    robot6axis/servo_4/StatusPosDecrease AT 182 : BOOL := false;
    robot6axis/servo_4/displayJauge AT 6454 : REAL := 0.0;
    robot6axis/servo_4/servo_mode/PLC_StatusReady AT 26 : BOOL := true;
    robot6axis/servo_4/servo_mode/PLC_StatusMoved AT 25 : BOOL := false;
    robot6axis/servo_4/servo_mode/PLC_StatusStand AT 24 : BOOL := false;
    robot6axis/servo_4/servo_mode/PLC_ActualPositionAx AT 161 : REAL := 0.0;
    robot6axis/servo_4/servo_mode/PLC_ActualPositionMa AT 48 : REAL := 0.0;
    robot6axis/servo_4/servo_mode/PLC_ActualVelocity AT 47 : REAL := 0.0;
    robot6axis/servo_4/servo_mode/StatusReady AT 266 : BOOL := true;
    robot6axis/servo_4/servo_mode/StatusMoved AT 267 : BOOL := false;
    robot6axis/servo_4/servo_mode/StatusStand AT 268 : BOOL := false;
    robot6axis/servo_4/servo_mode/ActualPositionMa AT 6824 : REAL := 0.0;
    robot6axis/servo_4/servo_mode/ActualVelocity AT 6825 : REAL := 0.0;
    robot6axis/servo_4/servo_mode/MaximumVelocity AT 6826 : REAL := 0.0;
    robot6axis/servo_4/servo_mode/physicalPosInit AT 6461 : REAL := 0.0;
    robot6axis/servo_4/servo_mode/ActualPositionAx AT 6463 : REAL := 0.0;
    robot6axis/servo_4/servo_mode/StatusReady_o AT 186 : BOOL := true;
    robot6axis/servo_4/servo_mode/StatusMoved_o AT 185 : BOOL := false;
    robot6axis/servo_4/servo_mode/StatusStand_o AT 184 : BOOL := false;
    robot6axis/servo_4/servo_mode/ActualPositionAx_o AT 6566 : REAL := 0.0;
    robot6axis/servo_4/servo_mode/ActualPositionMa_o AT 6456 : REAL := 0.0;
    robot6axis/servo_4/servo_mode/ActualVelocity_o AT 39 : REAL := 0.0;
    robot6axis/servo_4/servo_mode/MaximumVelocity_o AT 6455 : REAL := 0.0;
    robot6axis/servo_4/servo_mode/StatusPosIncrease_o AT 183 : BOOL := false;
    robot6axis/servo_4/servo_mode/StatusPosDecrease_o AT 182 : BOOL := false;
    robot6axis/servo_4/servo_mode/displayJauge_o AT 6454 : REAL := 0.0;
    robot6axis/servo_4/servo_mode/PLCMode AT 273 : BOOL := false;
    robot6axis/servo_4/servo_mode/PLCMode1 AT 274 : BOOL := false;
    robot6axis/servo_4/servo_mode/initDone AT 275 : BOOL := false;
    robot6axis/servo_4/servo_mode/displayPosMin AT 6829 : REAL := 0.0;
    robot6axis/servo_4/servo_mode/displayPosMax AT 6830 : REAL := 0.0;
    robot6axis/servo_4/servo_mode/PLC_ActualPositionAx1 AT 6831 : REAL := 0.0;
    robot6axis/servo_4/servo_mode/PLC_ActualVelocity1 AT 6832 : REAL := 0.0;
    robot6axis/servo_4/servo_mode/ActualPositionAx1 AT 6833 : REAL := 0.0;
    robot6axis/servo_4/servo_mode/ActualVelocity1 AT 6834 : REAL := 0.0;
    robot6axis/servo_4/servo_mode/offsetAxToMa AT 6835 : REAL := 0.0;
    robot6axis/servo_4/servo_mode/offsetAxToMa1 AT 6836 : REAL := 0.0;
    robot6axis/servo_4/servo_mode/ActualPositionMa_o1 AT 6837 : REAL := 0.0;
    robot6axis/servo_4/servo_control/HomeCmd AT 56 : BOOL := false;
    robot6axis/servo_4/servo_control/MoveVelCmd AT 55 : BOOL := false;
    robot6axis/servo_4/servo_control/MoveAbsCmd AT 54 : BOOL := false;
    robot6axis/servo_4/servo_control/MoveVel1ManualCmd AT 53 : BOOL := false;
    robot6axis/servo_4/servo_control/MoveVel2ManualCmd AT 52 : BOOL := false;
    robot6axis/servo_4/servo_control/MoveAbs1ManualCmd AT 51 : BOOL := false;
    robot6axis/servo_4/servo_control/MoveAbs2ManualCmd AT 50 : BOOL := false;
    robot6axis/servo_4/servo_control/StopCmd AT 14 : BOOL := false;
    robot6axis/servo_4/servo_control/MovePosition AT 69 : REAL := 0.0;
    robot6axis/servo_4/servo_control/MoveSpeed AT 68 : REAL := 100.0;
    robot6axis/servo_4/servo_control/MoveAcceleration AT 67 : REAL := 100.0;
    robot6axis/servo_4/servo_control/MoveDeceleration AT 66 : REAL := 100.0;
    robot6axis/servo_4/servo_control/offsetAxToMa AT 65 : REAL := 0.0;
    robot6axis/servo_4/servo_control/physicalPosInit AT 6461 : REAL := 0.0;
    robot6axis/servo_4/servo_control/MAX_SPEED AT 6460 : REAL(0.0..3.4e+038) := 30.0;
    robot6axis/servo_4/servo_control/status AT 621 : INT := 0;
    robot6axis/servo_4/servo_control/errorFlag AT 620 : INT := 0;
    robot6axis/servo_4/servo_control/IOActualPositionAx AT 6463 : REAL := 0.0;
    robot6axis/servo_4/servo_control/IOVelDone AT 188 : BOOL := false;
    robot6axis/servo_4/servo_control/IOAbsDone AT 187 : BOOL := false;
    robot6axis/servo_4/servo_control/IOActualVelocity AT 6462 : REAL := 0.0;
    robot6axis/servo_4/servo_control/OperationMode AT 655 : INT := 0;
    robot6axis/servo_4/servo_control/StatusReady AT 266 : BOOL := true;
    robot6axis/servo_4/servo_control/StatusMove AT 267 : BOOL := false;
    robot6axis/servo_4/servo_control/StatusStand AT 268 : BOOL := false;
    robot6axis/servo_4/servo_control/ActualPositionMa AT 6824 : REAL := 0.0;
    robot6axis/servo_4/servo_control/ActualVelocity AT 6825 : REAL := 0.0;
    robot6axis/servo_4/servo_control/MaximumVelocity AT 6826 : REAL := 0.0;
    robot6axis/servo_4/servo_control/VelEnabled AT 269 : BOOL := false;
    robot6axis/servo_4/servo_control/VelCmd AT 270 : BOOL := false;
    robot6axis/servo_4/servo_control/PosEnabled AT 271 : BOOL := false;
    robot6axis/servo_4/servo_control/PosCmd AT 272 : BOOL := false;
    robot6axis/servo_4/servo_control/Position AT 6828 : REAL := 0.0;
    robot6axis/servo_4/servo_control/Speed AT 6827 : REAL := 0.0;
    robot6axis/servo_4/servo_control/ManualMode AT 656 : INT := 0;
    robot6axis/servo_4/servo_control/initDone AT 276 : BOOL := false;
    robot6axis/servo_4/servo_control/ActualPositionMa1 AT 6838 : REAL := 0.0;
    robot6axis/servo_4/servo_control/offsetAxToMa1 AT 6839 : REAL := 0.0;
    robot6axis/servo_4/servo_control/HOME_POSITION AT 6840 : REAL := 100.0;
    robot6axis/servo_4/servo_control/MANUAL_POSITION1 AT 6841 : REAL := 0.0;
    robot6axis/servo_4/servo_control/MANUAL_POSITION2 AT 6842 : REAL := 150.0;
    robot6axis/servo_4/servo_control/MANUAL_SPEED1 AT 6843 : REAL := -100.0;
    robot6axis/servo_4/servo_control/MANUAL_SPEED2 AT 6844 : REAL := 100.0;
    robot6axis/servo_4/servo_control/MANUAL_SPEED AT 6845 : REAL := 100.0;
    robot6axis/servo_4/servo_velocity/MoveVelEnable AT 269 : BOOL := false;
    robot6axis/servo_4/servo_velocity/MoveVelStart AT 270 : BOOL := false;
    robot6axis/servo_4/servo_velocity/MoveSpeed AT 6827 : REAL := 0.0;
    robot6axis/servo_4/servo_velocity/MoveAcceleration AT 67 : REAL := 100.0;
    robot6axis/servo_4/servo_velocity/MoveDeceleration AT 66 : REAL := 100.0;
    robot6axis/servo_4/servo_velocity/MAX_SPEED AT 6460 : REAL(0.0..3.4e+038) := 30.0;
    robot6axis/servo_4/servo_velocity/MAX_ACCEL AT 6459 : REAL(0.0..3.4e+038) := 1500.0;
    robot6axis/servo_4/servo_velocity/MAX_DECEL AT 6458 : REAL(0.0..3.4e+038) := 1500.0;
    robot6axis/servo_4/servo_velocity/MODULO_LENGTH AT 6457 : REAL := 0.0;
    robot6axis/servo_4/servo_velocity/status AT 621 : INT := 0;
    robot6axis/servo_4/servo_velocity/errorFlag AT 620 : INT := 0;
    robot6axis/servo_4/servo_velocity/MoveVelDone AT 188 : BOOL := false;
    robot6axis/servo_4/servo_velocity/ActualPositionAx AT 6463 : REAL := 0.0;
    robot6axis/servo_4/servo_velocity/ActualVelocity AT 6462 : REAL := 0.0;
    robot6axis/servo_4/servo_velocity/firstStep AT 277 : BOOL := true;
    robot6axis/servo_4/servo_velocity/stepDone AT 278 : BOOL := false;
    robot6axis/servo_4/servo_velocity/currentTime AT 6846 : REAL := 0.0;
    robot6axis/servo_4/servo_velocity/MoveSpeed1 AT 6847 : REAL := 0.0;
    robot6axis/servo_4/servo_velocity/acceleration AT 6848 : REAL := 0.0;
    robot6axis/servo_4/servo_velocity/deceleration AT 6849 : REAL := 0.0;
    robot6axis/servo_4/servo_velocity/orderSpeed AT 6850 : REAL := 0.0;
    robot6axis/servo_4/servo_velocity/endChangeSpeed AT 6851 : REAL := 0.0;
    robot6axis/servo_4/servo_velocity/accelDecelChangeSpeed AT 6852 : REAL := 0.0;
    robot6axis/servo_4/servo_velocity/ActualVelocity1 AT 6853 : REAL := 0.0;
    robot6axis/servo_4/servo_velocity/speedChanged AT 279 : BOOL := false;
    robot6axis/servo_4/servo_position/MoveAbsEnable AT 271 : BOOL := false;
    robot6axis/servo_4/servo_position/MoveAbsStart AT 272 : BOOL := false;
    robot6axis/servo_4/servo_position/MovePosition AT 6828 : REAL := 0.0;
    robot6axis/servo_4/servo_position/MoveSpeed AT 6827 : REAL := 0.0;
    robot6axis/servo_4/servo_position/MoveAcceleration AT 67 : REAL := 100.0;
    robot6axis/servo_4/servo_position/MoveDeceleration AT 66 : REAL := 100.0;
    robot6axis/servo_4/servo_position/MAX_SPEED AT 6460 : REAL(0.0..3.4e+038) := 30.0;
    robot6axis/servo_4/servo_position/MAX_ACCEL AT 6459 : REAL(0.0..3.4e+038) := 1500.0;
    robot6axis/servo_4/servo_position/MAX_DECEL AT 6458 : REAL(0.0..3.4e+038) := 1500.0;
    robot6axis/servo_4/servo_position/MODULO_LENGTH AT 6457 : REAL := 0.0;
    robot6axis/servo_4/servo_position/status AT 621 : INT := 0;
    robot6axis/servo_4/servo_position/errorFlag AT 620 : INT := 0;
    robot6axis/servo_4/servo_position/MoveAbsDone AT 187 : BOOL := false;
    robot6axis/servo_4/servo_position/ActualPositionAx AT 6463 : REAL := 0.0;
    robot6axis/servo_4/servo_position/ActualVelocity AT 6462 : REAL := 0.0;
    robot6axis/servo_4/servo_position/firstStep AT 280 : BOOL := true;
    robot6axis/servo_4/servo_position/stepDone AT 281 : BOOL := false;
    robot6axis/servo_4/servo_position/timeToStop AT 6854 : REAL := 0.0;
    robot6axis/servo_4/servo_position/distanceToStop AT 6855 : REAL := 0.0;
    robot6axis/servo_4/servo_position/distance AT 6856 : REAL := 0.0;
    robot6axis/servo_4/servo_position/currentTime AT 6857 : REAL := 0.0;
    robot6axis/servo_4/servo_position/currentSpeed1 AT 6858 : REAL := 0.0;
    robot6axis/servo_4/servo_position/targetPosition AT 6859 : REAL := 0.0;
    robot6axis/servo_4/servo_position/ActualPositionAx1 AT 6860 : REAL := 0.0;
    robot6axis/servo_4/servo_position/acceleration AT 6861 : REAL := 0.0;
    robot6axis/servo_4/servo_position/deceleration AT 6862 : REAL := 0.0;
    robot6axis/servo_4/servo_position/orderSpeed AT 6863 : REAL := 0.0;
    robot6axis/servo_4/servo_position/moveDirection AT 6864 : REAL := 0.0;
    robot6axis/servo_4/servo_position/moveDirection1 AT 6865 : REAL := 0.0;
    robot6axis/servo_4/servo_position/endChangeSpeed AT 6866 : REAL := 0.0;
    robot6axis/servo_4/servo_position/ActualVelocity1 AT 6867 : REAL := 0.0;
    robot6axis/arm4/armOrigin AT 6555 : ARRAY[1..3] OF REAL := [3(0.0)];
    robot6axis/arm4/overallArmQuatInput AT 6560 : ARRAY[1..4] OF REAL := [4(0.0)];
    robot6axis/arm4/structRotVector AT 6449 : ARRAY[1..3] OF REAL := [2(0.0), 1.0];
    robot6axis/arm4/structRotDeg AT 6448 : REAL := 0.0;
    robot6axis/arm4/driveRotVector AT 119 : ARRAY[1..3] OF REAL := [1.0, 2(0.0)];
    robot6axis/arm4/driveRotDeg AT 6566 : REAL := 0.0;
    robot6axis/arm4/ownRotDeg AT 6447 : REAL := 0.0;
    robot6axis/arm4/driveResizeLength AT 6446 : REAL := 0.0;
    robot6axis/arm4/functionActive AT 181 : BOOL := false;
    robot6axis/arm4/armExtrem AT 6567 : ARRAY[1..3] OF REAL := [3(0.0)];
    robot6axis/arm4/overallArmRotOutput AT 6572 : ARRAY[1..4] OF REAL := [4(0.0)];
    robot6axis/arm4/productId AT 619 : DINT := -1;
    robot6axis/arm4/status_act_prod AT 657 : DINT := 0;
    robot6axis/arm4/m11 AT 6868 : REAL := 42.4403;
    robot6axis/arm4/m12 AT 6869 : REAL := 0.0;
    robot6axis/arm4/m13 AT 6870 : REAL := 0.0;
    robot6axis/arm4/m14 AT 6871 : REAL := 11.3174;
    robot6axis/arm4/m21 AT 6872 : REAL := 0.0;
    robot6axis/arm4/m22 AT 6873 : REAL := 31.1229;
    robot6axis/arm4/m23 AT 6874 : REAL := 0.0;
    robot6axis/arm4/m24 AT 6875 : REAL := 100.088;
    robot6axis/arm4/m31 AT 6876 : REAL := 0.0;
    robot6axis/arm4/m32 AT 6877 : REAL := 0.0;
    robot6axis/arm4/m33 AT 6878 : REAL := 9.90274;
    robot6axis/arm4/m34 AT 6879 : REAL := 10.6101;
    robot6axis/arm4/m41 AT 6880 : REAL := 0.0;
    robot6axis/arm4/m42 AT 6881 : REAL := 0.0;
    robot6axis/arm4/m43 AT 6882 : REAL := 0.0;
    robot6axis/arm4/m44 AT 6883 : REAL := 1.0;
    robot6axis/arm4/armLengthCalc AT 6884 : REAL := 0.0;
    robot6axis/arm4/functionActiveLocale AT 282 : BOOL := false;
    robot6axis/arm4/product_id AT 658 : DINT := -1;
    robot6axis/arm4/arm_id AT 659 : DINT := -1;
    robot6axis/arm4/timeToGripParam AT 6885 : REAL := 0.15;
    robot6axis/arm4/armLength AT 6886 : REAL := 202.0;
    robot6axis/arm4/armWidth AT 6887 : REAL := 40.0;
    robot6axis/arm4/armHeight AT 6888 : REAL := 40.0;
    robot6axis/arm4/armType AT 660 : INT := 0;
    robot6axis/servo_5/status AT 618 : INT := 0;
    robot6axis/servo_5/errorFlag AT 617 : INT := 0;
    robot6axis/servo_5/ActualPositionAx1 AT 6445 : REAL := 0.0;
    robot6axis/servo_5/MoveVelDone1 AT 180 : BOOL := false;
    robot6axis/servo_5/ActualVelocity1 AT 6444 : REAL := 0.0;
    robot6axis/servo_5/MoveAbsDone1 AT 179 : BOOL := false;
    robot6axis/servo_5/HomeCmd AT 49 : BOOL := false;
    robot6axis/servo_5/MoveVelCmd AT 48 : BOOL := false;
    robot6axis/servo_5/MoveAbsCmd AT 47 : BOOL := false;
    robot6axis/servo_5/MoveVel1ManualCmd AT 46 : BOOL := false;
    robot6axis/servo_5/MoveVel2ManualCmd AT 45 : BOOL := false;
    robot6axis/servo_5/MoveAbs1ManualCmd AT 44 : BOOL := false;
    robot6axis/servo_5/MoveAbs2ManualCmd AT 43 : BOOL := false;
    robot6axis/servo_5/StopCmd AT 14 : BOOL := false;
    robot6axis/servo_5/MovePosition AT 64 : REAL := 0.0;
    robot6axis/servo_5/MoveSpeed AT 63 : REAL := 100.0;
    robot6axis/servo_5/MoveAcceleration AT 62 : REAL := 100.0;
    robot6axis/servo_5/MoveDeceleration AT 61 : REAL := 100.0;
    robot6axis/servo_5/offsetAxToMa AT 60 : REAL := 0.0;
    robot6axis/servo_5/PLC_StatusReady AT 23 : BOOL := true;
    robot6axis/servo_5/PLC_StatusMoved AT 22 : BOOL := false;
    robot6axis/servo_5/PLC_StatusStand AT 21 : BOOL := false;
    robot6axis/servo_5/PLC_ActualPositionAx AT 162 : REAL := 0.0;
    robot6axis/servo_5/PLC_ActualPositionMa AT 46 : REAL := 0.0;
    robot6axis/servo_5/PLC_ActualVelocity AT 45 : REAL := 0.0;
    robot6axis/servo_5/physicalPosInit AT 6443 : REAL := 0.0;
    robot6axis/servo_5/MAX_SPEED AT 6442 : REAL(0.0..3.4e+038) := 30.0;
    robot6axis/servo_5/MAX_ACCEL AT 6441 : REAL(0.0..3.4e+038) := 1500.0;
    robot6axis/servo_5/MAX_DECEL AT 6440 : REAL(0.0..3.4e+038) := 1500.0;
    robot6axis/servo_5/MODULO_LENGTH AT 6439 : REAL := 0.0;
    robot6axis/servo_5/StatusReady AT 178 : BOOL := true;
    robot6axis/servo_5/StatusMoved AT 177 : BOOL := false;
    robot6axis/servo_5/StatusStand AT 176 : BOOL := false;
    robot6axis/servo_5/ActualPositionAx AT 6578 : REAL := 0.0;
    robot6axis/servo_5/ActualPositionMa AT 6438 : REAL := 0.0;
    robot6axis/servo_5/ActualVelocity AT 38 : REAL := 0.0;
    robot6axis/servo_5/MaximumVelocity AT 6437 : REAL := 0.0;
    robot6axis/servo_5/StatusPosIncrease AT 175 : BOOL := false;
    robot6axis/servo_5/StatusPosDecrease AT 174 : BOOL := false;
    robot6axis/servo_5/displayJauge AT 6436 : REAL := 0.0;
    robot6axis/servo_5/servo_mode/PLC_StatusReady AT 23 : BOOL := true;
    robot6axis/servo_5/servo_mode/PLC_StatusMoved AT 22 : BOOL := false;
    robot6axis/servo_5/servo_mode/PLC_StatusStand AT 21 : BOOL := false;
    robot6axis/servo_5/servo_mode/PLC_ActualPositionAx AT 162 : REAL := 0.0;
    robot6axis/servo_5/servo_mode/PLC_ActualPositionMa AT 46 : REAL := 0.0;
    robot6axis/servo_5/servo_mode/PLC_ActualVelocity AT 45 : REAL := 0.0;
    robot6axis/servo_5/servo_mode/StatusReady AT 283 : BOOL := true;
    robot6axis/servo_5/servo_mode/StatusMoved AT 284 : BOOL := false;
    robot6axis/servo_5/servo_mode/StatusStand AT 285 : BOOL := false;
    robot6axis/servo_5/servo_mode/ActualPositionMa AT 6889 : REAL := 0.0;
    robot6axis/servo_5/servo_mode/ActualVelocity AT 6890 : REAL := 0.0;
    robot6axis/servo_5/servo_mode/MaximumVelocity AT 6891 : REAL := 0.0;
    robot6axis/servo_5/servo_mode/physicalPosInit AT 6443 : REAL := 0.0;
    robot6axis/servo_5/servo_mode/ActualPositionAx AT 6445 : REAL := 0.0;
    robot6axis/servo_5/servo_mode/StatusReady_o AT 178 : BOOL := true;
    robot6axis/servo_5/servo_mode/StatusMoved_o AT 177 : BOOL := false;
    robot6axis/servo_5/servo_mode/StatusStand_o AT 176 : BOOL := false;
    robot6axis/servo_5/servo_mode/ActualPositionAx_o AT 6578 : REAL := 0.0;
    robot6axis/servo_5/servo_mode/ActualPositionMa_o AT 6438 : REAL := 0.0;
    robot6axis/servo_5/servo_mode/ActualVelocity_o AT 38 : REAL := 0.0;
    robot6axis/servo_5/servo_mode/MaximumVelocity_o AT 6437 : REAL := 0.0;
    robot6axis/servo_5/servo_mode/StatusPosIncrease_o AT 175 : BOOL := false;
    robot6axis/servo_5/servo_mode/StatusPosDecrease_o AT 174 : BOOL := false;
    robot6axis/servo_5/servo_mode/displayJauge_o AT 6436 : REAL := 0.0;
    robot6axis/servo_5/servo_mode/PLCMode AT 290 : BOOL := false;
    robot6axis/servo_5/servo_mode/PLCMode1 AT 291 : BOOL := false;
    robot6axis/servo_5/servo_mode/initDone AT 292 : BOOL := false;
    robot6axis/servo_5/servo_mode/displayPosMin AT 6894 : REAL := 0.0;
    robot6axis/servo_5/servo_mode/displayPosMax AT 6895 : REAL := 0.0;
    robot6axis/servo_5/servo_mode/PLC_ActualPositionAx1 AT 6896 : REAL := 0.0;
    robot6axis/servo_5/servo_mode/PLC_ActualVelocity1 AT 6897 : REAL := 0.0;
    robot6axis/servo_5/servo_mode/ActualPositionAx1 AT 6898 : REAL := 0.0;
    robot6axis/servo_5/servo_mode/ActualVelocity1 AT 6899 : REAL := 0.0;
    robot6axis/servo_5/servo_mode/offsetAxToMa AT 6900 : REAL := 0.0;
    robot6axis/servo_5/servo_mode/offsetAxToMa1 AT 6901 : REAL := 0.0;
    robot6axis/servo_5/servo_mode/ActualPositionMa_o1 AT 6902 : REAL := 0.0;
    robot6axis/servo_5/servo_control/HomeCmd AT 49 : BOOL := false;
    robot6axis/servo_5/servo_control/MoveVelCmd AT 48 : BOOL := false;
    robot6axis/servo_5/servo_control/MoveAbsCmd AT 47 : BOOL := false;
    robot6axis/servo_5/servo_control/MoveVel1ManualCmd AT 46 : BOOL := false;
    robot6axis/servo_5/servo_control/MoveVel2ManualCmd AT 45 : BOOL := false;
    robot6axis/servo_5/servo_control/MoveAbs1ManualCmd AT 44 : BOOL := false;
    robot6axis/servo_5/servo_control/MoveAbs2ManualCmd AT 43 : BOOL := false;
    robot6axis/servo_5/servo_control/StopCmd AT 14 : BOOL := false;
    robot6axis/servo_5/servo_control/MovePosition AT 64 : REAL := 0.0;
    robot6axis/servo_5/servo_control/MoveSpeed AT 63 : REAL := 100.0;
    robot6axis/servo_5/servo_control/MoveAcceleration AT 62 : REAL := 100.0;
    robot6axis/servo_5/servo_control/MoveDeceleration AT 61 : REAL := 100.0;
    robot6axis/servo_5/servo_control/offsetAxToMa AT 60 : REAL := 0.0;
    robot6axis/servo_5/servo_control/physicalPosInit AT 6443 : REAL := 0.0;
    robot6axis/servo_5/servo_control/MAX_SPEED AT 6442 : REAL(0.0..3.4e+038) := 30.0;
    robot6axis/servo_5/servo_control/status AT 618 : INT := 0;
    robot6axis/servo_5/servo_control/errorFlag AT 617 : INT := 0;
    robot6axis/servo_5/servo_control/IOActualPositionAx AT 6445 : REAL := 0.0;
    robot6axis/servo_5/servo_control/IOVelDone AT 180 : BOOL := false;
    robot6axis/servo_5/servo_control/IOAbsDone AT 179 : BOOL := false;
    robot6axis/servo_5/servo_control/IOActualVelocity AT 6444 : REAL := 0.0;
    robot6axis/servo_5/servo_control/OperationMode AT 661 : INT := 0;
    robot6axis/servo_5/servo_control/StatusReady AT 283 : BOOL := true;
    robot6axis/servo_5/servo_control/StatusMove AT 284 : BOOL := false;
    robot6axis/servo_5/servo_control/StatusStand AT 285 : BOOL := false;
    robot6axis/servo_5/servo_control/ActualPositionMa AT 6889 : REAL := 0.0;
    robot6axis/servo_5/servo_control/ActualVelocity AT 6890 : REAL := 0.0;
    robot6axis/servo_5/servo_control/MaximumVelocity AT 6891 : REAL := 0.0;
    robot6axis/servo_5/servo_control/VelEnabled AT 286 : BOOL := false;
    robot6axis/servo_5/servo_control/VelCmd AT 287 : BOOL := false;
    robot6axis/servo_5/servo_control/PosEnabled AT 288 : BOOL := false;
    robot6axis/servo_5/servo_control/PosCmd AT 289 : BOOL := false;
    robot6axis/servo_5/servo_control/Position AT 6893 : REAL := 0.0;
    robot6axis/servo_5/servo_control/Speed AT 6892 : REAL := 0.0;
    robot6axis/servo_5/servo_control/ManualMode AT 662 : INT := 0;
    robot6axis/servo_5/servo_control/initDone AT 293 : BOOL := false;
    robot6axis/servo_5/servo_control/ActualPositionMa1 AT 6903 : REAL := 0.0;
    robot6axis/servo_5/servo_control/offsetAxToMa1 AT 6904 : REAL := 0.0;
    robot6axis/servo_5/servo_control/HOME_POSITION AT 6905 : REAL := 100.0;
    robot6axis/servo_5/servo_control/MANUAL_POSITION1 AT 6906 : REAL := 0.0;
    robot6axis/servo_5/servo_control/MANUAL_POSITION2 AT 6907 : REAL := 150.0;
    robot6axis/servo_5/servo_control/MANUAL_SPEED1 AT 6908 : REAL := -100.0;
    robot6axis/servo_5/servo_control/MANUAL_SPEED2 AT 6909 : REAL := 100.0;
    robot6axis/servo_5/servo_control/MANUAL_SPEED AT 6910 : REAL := 100.0;
    robot6axis/servo_5/servo_velocity/MoveVelEnable AT 286 : BOOL := false;
    robot6axis/servo_5/servo_velocity/MoveVelStart AT 287 : BOOL := false;
    robot6axis/servo_5/servo_velocity/MoveSpeed AT 6892 : REAL := 0.0;
    robot6axis/servo_5/servo_velocity/MoveAcceleration AT 62 : REAL := 100.0;
    robot6axis/servo_5/servo_velocity/MoveDeceleration AT 61 : REAL := 100.0;
    robot6axis/servo_5/servo_velocity/MAX_SPEED AT 6442 : REAL(0.0..3.4e+038) := 30.0;
    robot6axis/servo_5/servo_velocity/MAX_ACCEL AT 6441 : REAL(0.0..3.4e+038) := 1500.0;
    robot6axis/servo_5/servo_velocity/MAX_DECEL AT 6440 : REAL(0.0..3.4e+038) := 1500.0;
    robot6axis/servo_5/servo_velocity/MODULO_LENGTH AT 6439 : REAL := 0.0;
    robot6axis/servo_5/servo_velocity/status AT 618 : INT := 0;
    robot6axis/servo_5/servo_velocity/errorFlag AT 617 : INT := 0;
    robot6axis/servo_5/servo_velocity/MoveVelDone AT 180 : BOOL := false;
    robot6axis/servo_5/servo_velocity/ActualPositionAx AT 6445 : REAL := 0.0;
    robot6axis/servo_5/servo_velocity/ActualVelocity AT 6444 : REAL := 0.0;
    robot6axis/servo_5/servo_velocity/firstStep AT 294 : BOOL := true;
    robot6axis/servo_5/servo_velocity/stepDone AT 295 : BOOL := false;
    robot6axis/servo_5/servo_velocity/currentTime AT 6911 : REAL := 0.0;
    robot6axis/servo_5/servo_velocity/MoveSpeed1 AT 6912 : REAL := 0.0;
    robot6axis/servo_5/servo_velocity/acceleration AT 6913 : REAL := 0.0;
    robot6axis/servo_5/servo_velocity/deceleration AT 6914 : REAL := 0.0;
    robot6axis/servo_5/servo_velocity/orderSpeed AT 6915 : REAL := 0.0;
    robot6axis/servo_5/servo_velocity/endChangeSpeed AT 6916 : REAL := 0.0;
    robot6axis/servo_5/servo_velocity/accelDecelChangeSpeed AT 6917 : REAL := 0.0;
    robot6axis/servo_5/servo_velocity/ActualVelocity1 AT 6918 : REAL := 0.0;
    robot6axis/servo_5/servo_velocity/speedChanged AT 296 : BOOL := false;
    robot6axis/servo_5/servo_position/MoveAbsEnable AT 288 : BOOL := false;
    robot6axis/servo_5/servo_position/MoveAbsStart AT 289 : BOOL := false;
    robot6axis/servo_5/servo_position/MovePosition AT 6893 : REAL := 0.0;
    robot6axis/servo_5/servo_position/MoveSpeed AT 6892 : REAL := 0.0;
    robot6axis/servo_5/servo_position/MoveAcceleration AT 62 : REAL := 100.0;
    robot6axis/servo_5/servo_position/MoveDeceleration AT 61 : REAL := 100.0;
    robot6axis/servo_5/servo_position/MAX_SPEED AT 6442 : REAL(0.0..3.4e+038) := 30.0;
    robot6axis/servo_5/servo_position/MAX_ACCEL AT 6441 : REAL(0.0..3.4e+038) := 1500.0;
    robot6axis/servo_5/servo_position/MAX_DECEL AT 6440 : REAL(0.0..3.4e+038) := 1500.0;
    robot6axis/servo_5/servo_position/MODULO_LENGTH AT 6439 : REAL := 0.0;
    robot6axis/servo_5/servo_position/status AT 618 : INT := 0;
    robot6axis/servo_5/servo_position/errorFlag AT 617 : INT := 0;
    robot6axis/servo_5/servo_position/MoveAbsDone AT 179 : BOOL := false;
    robot6axis/servo_5/servo_position/ActualPositionAx AT 6445 : REAL := 0.0;
    robot6axis/servo_5/servo_position/ActualVelocity AT 6444 : REAL := 0.0;
    robot6axis/servo_5/servo_position/firstStep AT 297 : BOOL := true;
    robot6axis/servo_5/servo_position/stepDone AT 298 : BOOL := false;
    robot6axis/servo_5/servo_position/timeToStop AT 6919 : REAL := 0.0;
    robot6axis/servo_5/servo_position/distanceToStop AT 6920 : REAL := 0.0;
    robot6axis/servo_5/servo_position/distance AT 6921 : REAL := 0.0;
    robot6axis/servo_5/servo_position/currentTime AT 6922 : REAL := 0.0;
    robot6axis/servo_5/servo_position/currentSpeed1 AT 6923 : REAL := 0.0;
    robot6axis/servo_5/servo_position/targetPosition AT 6924 : REAL := 0.0;
    robot6axis/servo_5/servo_position/ActualPositionAx1 AT 6925 : REAL := 0.0;
    robot6axis/servo_5/servo_position/acceleration AT 6926 : REAL := 0.0;
    robot6axis/servo_5/servo_position/deceleration AT 6927 : REAL := 0.0;
    robot6axis/servo_5/servo_position/orderSpeed AT 6928 : REAL := 0.0;
    robot6axis/servo_5/servo_position/moveDirection AT 6929 : REAL := 0.0;
    robot6axis/servo_5/servo_position/moveDirection1 AT 6930 : REAL := 0.0;
    robot6axis/servo_5/servo_position/endChangeSpeed AT 6931 : REAL := 0.0;
    robot6axis/servo_5/servo_position/ActualVelocity1 AT 6932 : REAL := 0.0;
    robot6axis/arm5/armOrigin AT 6567 : ARRAY[1..3] OF REAL := [3(0.0)];
    robot6axis/arm5/overallArmQuatInput AT 6572 : ARRAY[1..4] OF REAL := [4(0.0)];
    robot6axis/arm5/structRotVector AT 6431 : ARRAY[1..3] OF REAL := [2(0.0), 1.0];
    robot6axis/arm5/structRotDeg AT 6430 : REAL := 0.0;
    robot6axis/arm5/driveRotVector AT 114 : ARRAY[1..3] OF REAL := [0.0, 1.0, 0.0];
    robot6axis/arm5/driveRotDeg AT 6578 : REAL := 0.0;
    robot6axis/arm5/ownRotDeg AT 6429 : REAL := 0.0;
    robot6axis/arm5/driveResizeLength AT 6428 : REAL := 0.0;
    robot6axis/arm5/functionActive AT 173 : BOOL := false;
    robot6axis/arm5/armExtrem AT 6579 : ARRAY[1..3] OF REAL := [3(0.0)];
    robot6axis/arm5/overallArmRotOutput AT 6584 : ARRAY[1..4] OF REAL := [4(0.0)];
    robot6axis/arm5/productId AT 616 : DINT := -1;
    robot6axis/arm5/status_act_prod AT 663 : DINT := 0;
    robot6axis/arm5/m11 AT 6933 : REAL := 38.1963;
    robot6axis/arm5/m12 AT 6934 : REAL := 0.0;
    robot6axis/arm5/m13 AT 6935 : REAL := 0.0;
    robot6axis/arm5/m14 AT 6936 : REAL := 8.48806;
    robot6axis/arm5/m21 AT 6937 : REAL := 0.0;
    robot6axis/arm5/m22 AT 6938 : REAL := 1.0;
    robot6axis/arm5/m23 AT 6939 : REAL := 0.0;
    robot6axis/arm5/m24 AT 6940 : REAL := 1.0;
    robot6axis/arm5/m31 AT 6941 : REAL := 0.0;
    robot6axis/arm5/m32 AT 6942 : REAL := 0.0;
    robot6axis/arm5/m33 AT 6943 : REAL := 14.1468;
    robot6axis/arm5/m34 AT 6944 : REAL := -10.6101;
    robot6axis/arm5/m41 AT 6945 : REAL := 0.0;
    robot6axis/arm5/m42 AT 6946 : REAL := 0.0;
    robot6axis/arm5/m43 AT 6947 : REAL := 0.0;
    robot6axis/arm5/m44 AT 6948 : REAL := 1.0;
    robot6axis/arm5/armLengthCalc AT 6949 : REAL := 0.0;
    robot6axis/arm5/functionActiveLocale AT 299 : BOOL := false;
    robot6axis/arm5/product_id AT 664 : DINT := -1;
    robot6axis/arm5/arm_id AT 665 : DINT := -1;
    robot6axis/arm5/timeToGripParam AT 6950 : REAL := 0.15;
    robot6axis/arm5/armLength AT 6951 : REAL := 61.0;
    robot6axis/arm5/armWidth AT 6952 : REAL := 40.0;
    robot6axis/arm5/armHeight AT 6953 : REAL := 40.0;
    robot6axis/arm5/armType AT 666 : INT := 0;
    robot6axis/servo_6/status AT 615 : INT := 0;
    robot6axis/servo_6/errorFlag AT 614 : INT := 0;
    robot6axis/servo_6/ActualPositionAx1 AT 6427 : REAL := 0.0;
    robot6axis/servo_6/MoveVelDone1 AT 172 : BOOL := false;
    robot6axis/servo_6/ActualVelocity1 AT 6426 : REAL := 0.0;
    robot6axis/servo_6/MoveAbsDone1 AT 171 : BOOL := false;
    robot6axis/servo_6/HomeCmd AT 42 : BOOL := false;
    robot6axis/servo_6/MoveVelCmd AT 41 : BOOL := false;
    robot6axis/servo_6/MoveAbsCmd AT 40 : BOOL := false;
    robot6axis/servo_6/MoveVel1ManualCmd AT 39 : BOOL := false;
    robot6axis/servo_6/MoveVel2ManualCmd AT 38 : BOOL := false;
    robot6axis/servo_6/MoveAbs1ManualCmd AT 37 : BOOL := false;
    robot6axis/servo_6/MoveAbs2ManualCmd AT 36 : BOOL := false;
    robot6axis/servo_6/StopCmd AT 14 : BOOL := false;
    robot6axis/servo_6/MovePosition AT 59 : REAL := 0.0;
    robot6axis/servo_6/MoveSpeed AT 58 : REAL := 100.0;
    robot6axis/servo_6/MoveAcceleration AT 57 : REAL := 100.0;
    robot6axis/servo_6/MoveDeceleration AT 56 : REAL := 100.0;
    robot6axis/servo_6/offsetAxToMa AT 55 : REAL := 0.0;
    robot6axis/servo_6/PLC_StatusReady AT 20 : BOOL := true;
    robot6axis/servo_6/PLC_StatusMoved AT 19 : BOOL := false;
    robot6axis/servo_6/PLC_StatusStand AT 18 : BOOL := false;
    robot6axis/servo_6/PLC_ActualPositionAx AT 163 : REAL := 0.0;
    robot6axis/servo_6/PLC_ActualPositionMa AT 44 : REAL := 0.0;
    robot6axis/servo_6/PLC_ActualVelocity AT 43 : REAL := 0.0;
    robot6axis/servo_6/physicalPosInit AT 6425 : REAL := 0.0;
    robot6axis/servo_6/MAX_SPEED AT 6424 : REAL(0.0..3.4e+038) := 30.0;
    robot6axis/servo_6/MAX_ACCEL AT 6423 : REAL(0.0..3.4e+038) := 1500.0;
    robot6axis/servo_6/MAX_DECEL AT 6422 : REAL(0.0..3.4e+038) := 1500.0;
    robot6axis/servo_6/MODULO_LENGTH AT 6421 : REAL := 0.0;
    robot6axis/servo_6/StatusReady AT 170 : BOOL := true;
    robot6axis/servo_6/StatusMoved AT 169 : BOOL := false;
    robot6axis/servo_6/StatusStand AT 168 : BOOL := false;
    robot6axis/servo_6/ActualPositionAx AT 6590 : REAL := 0.0;
    robot6axis/servo_6/ActualPositionMa AT 6420 : REAL := 0.0;
    robot6axis/servo_6/ActualVelocity AT 37 : REAL := 0.0;
    robot6axis/servo_6/MaximumVelocity AT 6419 : REAL := 0.0;
    robot6axis/servo_6/StatusPosIncrease AT 167 : BOOL := false;
    robot6axis/servo_6/StatusPosDecrease AT 166 : BOOL := false;
    robot6axis/servo_6/displayJauge AT 6418 : REAL := 0.0;
    robot6axis/servo_6/servo_mode/PLC_StatusReady AT 20 : BOOL := true;
    robot6axis/servo_6/servo_mode/PLC_StatusMoved AT 19 : BOOL := false;
    robot6axis/servo_6/servo_mode/PLC_StatusStand AT 18 : BOOL := false;
    robot6axis/servo_6/servo_mode/PLC_ActualPositionAx AT 163 : REAL := 0.0;
    robot6axis/servo_6/servo_mode/PLC_ActualPositionMa AT 44 : REAL := 0.0;
    robot6axis/servo_6/servo_mode/PLC_ActualVelocity AT 43 : REAL := 0.0;
    robot6axis/servo_6/servo_mode/StatusReady AT 300 : BOOL := true;
    robot6axis/servo_6/servo_mode/StatusMoved AT 301 : BOOL := false;
    robot6axis/servo_6/servo_mode/StatusStand AT 302 : BOOL := false;
    robot6axis/servo_6/servo_mode/ActualPositionMa AT 6954 : REAL := 0.0;
    robot6axis/servo_6/servo_mode/ActualVelocity AT 6955 : REAL := 0.0;
    robot6axis/servo_6/servo_mode/MaximumVelocity AT 6956 : REAL := 0.0;
    robot6axis/servo_6/servo_mode/physicalPosInit AT 6425 : REAL := 0.0;
    robot6axis/servo_6/servo_mode/ActualPositionAx AT 6427 : REAL := 0.0;
    robot6axis/servo_6/servo_mode/StatusReady_o AT 170 : BOOL := true;
    robot6axis/servo_6/servo_mode/StatusMoved_o AT 169 : BOOL := false;
    robot6axis/servo_6/servo_mode/StatusStand_o AT 168 : BOOL := false;
    robot6axis/servo_6/servo_mode/ActualPositionAx_o AT 6590 : REAL := 0.0;
    robot6axis/servo_6/servo_mode/ActualPositionMa_o AT 6420 : REAL := 0.0;
    robot6axis/servo_6/servo_mode/ActualVelocity_o AT 37 : REAL := 0.0;
    robot6axis/servo_6/servo_mode/MaximumVelocity_o AT 6419 : REAL := 0.0;
    robot6axis/servo_6/servo_mode/StatusPosIncrease_o AT 167 : BOOL := false;
    robot6axis/servo_6/servo_mode/StatusPosDecrease_o AT 166 : BOOL := false;
    robot6axis/servo_6/servo_mode/displayJauge_o AT 6418 : REAL := 0.0;
    robot6axis/servo_6/servo_mode/PLCMode AT 307 : BOOL := false;
    robot6axis/servo_6/servo_mode/PLCMode1 AT 308 : BOOL := false;
    robot6axis/servo_6/servo_mode/initDone AT 309 : BOOL := false;
    robot6axis/servo_6/servo_mode/displayPosMin AT 6959 : REAL := 0.0;
    robot6axis/servo_6/servo_mode/displayPosMax AT 6960 : REAL := 0.0;
    robot6axis/servo_6/servo_mode/PLC_ActualPositionAx1 AT 6961 : REAL := 0.0;
    robot6axis/servo_6/servo_mode/PLC_ActualVelocity1 AT 6962 : REAL := 0.0;
    robot6axis/servo_6/servo_mode/ActualPositionAx1 AT 6963 : REAL := 0.0;
    robot6axis/servo_6/servo_mode/ActualVelocity1 AT 6964 : REAL := 0.0;
    robot6axis/servo_6/servo_mode/offsetAxToMa AT 6965 : REAL := 0.0;
    robot6axis/servo_6/servo_mode/offsetAxToMa1 AT 6966 : REAL := 0.0;
    robot6axis/servo_6/servo_mode/ActualPositionMa_o1 AT 6967 : REAL := 0.0;
    robot6axis/servo_6/servo_control/HomeCmd AT 42 : BOOL := false;
    robot6axis/servo_6/servo_control/MoveVelCmd AT 41 : BOOL := false;
    robot6axis/servo_6/servo_control/MoveAbsCmd AT 40 : BOOL := false;
    robot6axis/servo_6/servo_control/MoveVel1ManualCmd AT 39 : BOOL := false;
    robot6axis/servo_6/servo_control/MoveVel2ManualCmd AT 38 : BOOL := false;
    robot6axis/servo_6/servo_control/MoveAbs1ManualCmd AT 37 : BOOL := false;
    robot6axis/servo_6/servo_control/MoveAbs2ManualCmd AT 36 : BOOL := false;
    robot6axis/servo_6/servo_control/StopCmd AT 14 : BOOL := false;
    robot6axis/servo_6/servo_control/MovePosition AT 59 : REAL := 0.0;
    robot6axis/servo_6/servo_control/MoveSpeed AT 58 : REAL := 100.0;
    robot6axis/servo_6/servo_control/MoveAcceleration AT 57 : REAL := 100.0;
    robot6axis/servo_6/servo_control/MoveDeceleration AT 56 : REAL := 100.0;
    robot6axis/servo_6/servo_control/offsetAxToMa AT 55 : REAL := 0.0;
    robot6axis/servo_6/servo_control/physicalPosInit AT 6425 : REAL := 0.0;
    robot6axis/servo_6/servo_control/MAX_SPEED AT 6424 : REAL(0.0..3.4e+038) := 30.0;
    robot6axis/servo_6/servo_control/status AT 615 : INT := 0;
    robot6axis/servo_6/servo_control/errorFlag AT 614 : INT := 0;
    robot6axis/servo_6/servo_control/IOActualPositionAx AT 6427 : REAL := 0.0;
    robot6axis/servo_6/servo_control/IOVelDone AT 172 : BOOL := false;
    robot6axis/servo_6/servo_control/IOAbsDone AT 171 : BOOL := false;
    robot6axis/servo_6/servo_control/IOActualVelocity AT 6426 : REAL := 0.0;
    robot6axis/servo_6/servo_control/OperationMode AT 667 : INT := 0;
    robot6axis/servo_6/servo_control/StatusReady AT 300 : BOOL := true;
    robot6axis/servo_6/servo_control/StatusMove AT 301 : BOOL := false;
    robot6axis/servo_6/servo_control/StatusStand AT 302 : BOOL := false;
    robot6axis/servo_6/servo_control/ActualPositionMa AT 6954 : REAL := 0.0;
    robot6axis/servo_6/servo_control/ActualVelocity AT 6955 : REAL := 0.0;
    robot6axis/servo_6/servo_control/MaximumVelocity AT 6956 : REAL := 0.0;
    robot6axis/servo_6/servo_control/VelEnabled AT 303 : BOOL := false;
    robot6axis/servo_6/servo_control/VelCmd AT 304 : BOOL := false;
    robot6axis/servo_6/servo_control/PosEnabled AT 305 : BOOL := false;
    robot6axis/servo_6/servo_control/PosCmd AT 306 : BOOL := false;
    robot6axis/servo_6/servo_control/Position AT 6958 : REAL := 0.0;
    robot6axis/servo_6/servo_control/Speed AT 6957 : REAL := 0.0;
    robot6axis/servo_6/servo_control/ManualMode AT 668 : INT := 0;
    robot6axis/servo_6/servo_control/initDone AT 310 : BOOL := false;
    robot6axis/servo_6/servo_control/ActualPositionMa1 AT 6968 : REAL := 0.0;
    robot6axis/servo_6/servo_control/offsetAxToMa1 AT 6969 : REAL := 0.0;
    robot6axis/servo_6/servo_control/HOME_POSITION AT 6970 : REAL := 100.0;
    robot6axis/servo_6/servo_control/MANUAL_POSITION1 AT 6971 : REAL := 0.0;
    robot6axis/servo_6/servo_control/MANUAL_POSITION2 AT 6972 : REAL := 150.0;
    robot6axis/servo_6/servo_control/MANUAL_SPEED1 AT 6973 : REAL := -100.0;
    robot6axis/servo_6/servo_control/MANUAL_SPEED2 AT 6974 : REAL := 100.0;
    robot6axis/servo_6/servo_control/MANUAL_SPEED AT 6975 : REAL := 100.0;
    robot6axis/servo_6/servo_velocity/MoveVelEnable AT 303 : BOOL := false;
    robot6axis/servo_6/servo_velocity/MoveVelStart AT 304 : BOOL := false;
    robot6axis/servo_6/servo_velocity/MoveSpeed AT 6957 : REAL := 0.0;
    robot6axis/servo_6/servo_velocity/MoveAcceleration AT 57 : REAL := 100.0;
    robot6axis/servo_6/servo_velocity/MoveDeceleration AT 56 : REAL := 100.0;
    robot6axis/servo_6/servo_velocity/MAX_SPEED AT 6424 : REAL(0.0..3.4e+038) := 30.0;
    robot6axis/servo_6/servo_velocity/MAX_ACCEL AT 6423 : REAL(0.0..3.4e+038) := 1500.0;
    robot6axis/servo_6/servo_velocity/MAX_DECEL AT 6422 : REAL(0.0..3.4e+038) := 1500.0;
    robot6axis/servo_6/servo_velocity/MODULO_LENGTH AT 6421 : REAL := 0.0;
    robot6axis/servo_6/servo_velocity/status AT 615 : INT := 0;
    robot6axis/servo_6/servo_velocity/errorFlag AT 614 : INT := 0;
    robot6axis/servo_6/servo_velocity/MoveVelDone AT 172 : BOOL := false;
    robot6axis/servo_6/servo_velocity/ActualPositionAx AT 6427 : REAL := 0.0;
    robot6axis/servo_6/servo_velocity/ActualVelocity AT 6426 : REAL := 0.0;
    robot6axis/servo_6/servo_velocity/firstStep AT 311 : BOOL := true;
    robot6axis/servo_6/servo_velocity/stepDone AT 312 : BOOL := false;
    robot6axis/servo_6/servo_velocity/currentTime AT 6976 : REAL := 0.0;
    robot6axis/servo_6/servo_velocity/MoveSpeed1 AT 6977 : REAL := 0.0;
    robot6axis/servo_6/servo_velocity/acceleration AT 6978 : REAL := 0.0;
    robot6axis/servo_6/servo_velocity/deceleration AT 6979 : REAL := 0.0;
    robot6axis/servo_6/servo_velocity/orderSpeed AT 6980 : REAL := 0.0;
    robot6axis/servo_6/servo_velocity/endChangeSpeed AT 6981 : REAL := 0.0;
    robot6axis/servo_6/servo_velocity/accelDecelChangeSpeed AT 6982 : REAL := 0.0;
    robot6axis/servo_6/servo_velocity/ActualVelocity1 AT 6983 : REAL := 0.0;
    robot6axis/servo_6/servo_velocity/speedChanged AT 313 : BOOL := false;
    robot6axis/servo_6/servo_position/MoveAbsEnable AT 305 : BOOL := false;
    robot6axis/servo_6/servo_position/MoveAbsStart AT 306 : BOOL := false;
    robot6axis/servo_6/servo_position/MovePosition AT 6958 : REAL := 0.0;
    robot6axis/servo_6/servo_position/MoveSpeed AT 6957 : REAL := 0.0;
    robot6axis/servo_6/servo_position/MoveAcceleration AT 57 : REAL := 100.0;
    robot6axis/servo_6/servo_position/MoveDeceleration AT 56 : REAL := 100.0;
    robot6axis/servo_6/servo_position/MAX_SPEED AT 6424 : REAL(0.0..3.4e+038) := 30.0;
    robot6axis/servo_6/servo_position/MAX_ACCEL AT 6423 : REAL(0.0..3.4e+038) := 1500.0;
    robot6axis/servo_6/servo_position/MAX_DECEL AT 6422 : REAL(0.0..3.4e+038) := 1500.0;
    robot6axis/servo_6/servo_position/MODULO_LENGTH AT 6421 : REAL := 0.0;
    robot6axis/servo_6/servo_position/status AT 615 : INT := 0;
    robot6axis/servo_6/servo_position/errorFlag AT 614 : INT := 0;
    robot6axis/servo_6/servo_position/MoveAbsDone AT 171 : BOOL := false;
    robot6axis/servo_6/servo_position/ActualPositionAx AT 6427 : REAL := 0.0;
    robot6axis/servo_6/servo_position/ActualVelocity AT 6426 : REAL := 0.0;
    robot6axis/servo_6/servo_position/firstStep AT 314 : BOOL := true;
    robot6axis/servo_6/servo_position/stepDone AT 315 : BOOL := false;
    robot6axis/servo_6/servo_position/timeToStop AT 6984 : REAL := 0.0;
    robot6axis/servo_6/servo_position/distanceToStop AT 6985 : REAL := 0.0;
    robot6axis/servo_6/servo_position/distance AT 6986 : REAL := 0.0;
    robot6axis/servo_6/servo_position/currentTime AT 6987 : REAL := 0.0;
    robot6axis/servo_6/servo_position/currentSpeed1 AT 6988 : REAL := 0.0;
    robot6axis/servo_6/servo_position/targetPosition AT 6989 : REAL := 0.0;
    robot6axis/servo_6/servo_position/ActualPositionAx1 AT 6990 : REAL := 0.0;
    robot6axis/servo_6/servo_position/acceleration AT 6991 : REAL := 0.0;
    robot6axis/servo_6/servo_position/deceleration AT 6992 : REAL := 0.0;
    robot6axis/servo_6/servo_position/orderSpeed AT 6993 : REAL := 0.0;
    robot6axis/servo_6/servo_position/moveDirection AT 6994 : REAL := 0.0;
    robot6axis/servo_6/servo_position/moveDirection1 AT 6995 : REAL := 0.0;
    robot6axis/servo_6/servo_position/endChangeSpeed AT 6996 : REAL := 0.0;
    robot6axis/servo_6/servo_position/ActualVelocity1 AT 6997 : REAL := 0.0;
    robot6axis/arm6/armOrigin AT 6579 : ARRAY[1..3] OF REAL := [3(0.0)];
    robot6axis/arm6/overallArmQuatInput AT 6584 : ARRAY[1..4] OF REAL := [4(0.0)];
    robot6axis/arm6/structRotVector AT 6413 : ARRAY[1..3] OF REAL := [2(0.0), 1.0];
    robot6axis/arm6/structRotDeg AT 6412 : REAL := 0.0;
    robot6axis/arm6/driveRotVector AT 109 : ARRAY[1..3] OF REAL := [1.0, 2(0.0)];
    robot6axis/arm6/driveRotDeg AT 6590 : REAL := 0.0;
    robot6axis/arm6/ownRotDeg AT 6411 : REAL := 0.0;
    robot6axis/arm6/driveResizeLength AT 6410 : REAL := 0.0;
    robot6axis/arm6/functionActive AT 165 : BOOL := false;
    robot6axis/arm6/armExtrem AT 27 : ARRAY[1..3] OF REAL := [3(0.0)];
    robot6axis/arm6/overallArmRotOutput AT 6591 : ARRAY[1..4] OF REAL := [4(0.0)];
    robot6axis/arm6/productId AT 632 : DINT := -1;
    robot6axis/arm6/status_act_prod AT 669 : DINT := 0;
    robot6axis/arm6/m11 AT 6998 : REAL := 38.1963;
    robot6axis/arm6/m12 AT 6999 : REAL := 0.0;
    robot6axis/arm6/m13 AT 7000 : REAL := 0.0;
    robot6axis/arm6/m14 AT 7001 : REAL := 12.7321;
    robot6axis/arm6/m21 AT 7002 : REAL := 0.0;
    robot6axis/arm6/m22 AT 7003 : REAL := 1.0;
    robot6axis/arm6/m23 AT 7004 : REAL := 0.0;
    robot6axis/arm6/m24 AT 7005 : REAL := 1.0;
    robot6axis/arm6/m31 AT 7006 : REAL := 0.0;
    robot6axis/arm6/m32 AT 7007 : REAL := 0.0;
    robot6axis/arm6/m33 AT 7008 : REAL := 12.7321;
    robot6axis/arm6/m34 AT 7009 : REAL := -30.4156;
    robot6axis/arm6/m41 AT 7010 : REAL := 0.0;
    robot6axis/arm6/m42 AT 7011 : REAL := 0.0;
    robot6axis/arm6/m43 AT 7012 : REAL := 0.0;
    robot6axis/arm6/m44 AT 7013 : REAL := 1.0;
    robot6axis/arm6/armLengthCalc AT 7014 : REAL := 0.0;
    robot6axis/arm6/functionActiveLocale AT 316 : BOOL := false;
    robot6axis/arm6/product_id AT 670 : DINT := -1;
    robot6axis/arm6/arm_id AT 671 : DINT := -1;
    robot6axis/arm6/timeToGripParam AT 7015 : REAL := 0.15;
    robot6axis/arm6/armLength AT 7016 : REAL := 9.0;
    robot6axis/arm6/armWidth AT 7017 : REAL := 5.0;
    robot6axis/arm6/armHeight AT 7018 : REAL := 5.0;
    robot6axis/arm6/armType AT 672 : INT := 0;
    robot6axis/function_trigger/armExtrem AT 27 : ARRAY[1..3] OF REAL := [3(0.0)];
    robot6axis/function_trigger/productId AT 632 : DINT := -1;
    robot6axis/function_trigger/velX AT 32 : REAL := 0.0;
    robot6axis/function_trigger/velY AT 33 : REAL := 0.0;
    robot6axis/function_trigger/velZ AT 34 : REAL := 0.0;
    robot6axis/function_trigger/armInStop AT 17 : BOOL := false;
    robot6axis/function_trigger/armExtrem1 AT 7019 : ARRAY[1..3] OF REAL := [3(0.0)];
    robot6axis/function_trigger/i AT 673 : INT := 0;
    robot6axis/function_trigger/productTimeDetect AT 7024 : REAL := 0.0;
    robot6axis/function_trigger/productDetected AT 317 : BOOL := false;
    robot6axis/function_trigger/productId1 AT 674 : DINT := -1;
    robot6axis/function_trigger/actionTake AT 318 : BOOL := false;
    robot6axis/function_trigger/activeArea AT 319 : BOOL := false;
    robot6axis/function_trigger/ACTIVE_AREA_Z AT 7025 : REAL := 1100.0;
    robot6axis/function_trigger/TEMPO_DETECTION_PRO AT 7026 : REAL := 0.2;
    robot6axis/arm1RowA/armOrigin AT 27 : ARRAY[1..3] OF REAL := [3(0.0)];
    robot6axis/arm1RowA/overallArmQuatInput AT 6591 : ARRAY[1..4] OF REAL := [4(0.0)];
    robot6axis/arm1RowA/structRotVector AT 104 : ARRAY[1..3] OF REAL := [0.0, 1.0, 0.0];
    robot6axis/arm1RowA/structRotDeg AT 103 : REAL := -90.0;
    robot6axis/arm1RowA/driveRotVector AT 6405 : ARRAY[1..3] OF REAL := [2(0.0), 1.0];
    robot6axis/arm1RowA/driveRotDeg AT 6404 : REAL := 0.0;
    robot6axis/arm1RowA/ownRotDeg AT 6403 : REAL := 0.0;
    robot6axis/arm1RowA/driveResizeLength AT 6402 : REAL := 0.0;
    robot6axis/arm1RowA/functionActive AT 164 : BOOL := false;
    robot6axis/arm1RowA/armExtrem AT 6597 : ARRAY[1..3] OF REAL := [3(0.0)];
    robot6axis/arm1RowA/overallArmRotOutput AT 6602 : ARRAY[1..4] OF REAL := [4(0.0)];
    robot6axis/arm1RowA/productId AT 613 : DINT := -1;
    robot6axis/arm1RowA/status_act_prod AT 675 : DINT := 0;
    robot6axis/arm1RowA/m11 AT 7027 : REAL := 53.7577;
    robot6axis/arm1RowA/m12 AT 7028 : REAL := 0.0;
    robot6axis/arm1RowA/m13 AT 7029 : REAL := 0.0;
    robot6axis/arm1RowA/m14 AT 7030 : REAL := 11.3174;
    robot6axis/arm1RowA/m21 AT 7031 : REAL := 0.0;
    robot6axis/arm1RowA/m22 AT 7032 : REAL := 1.0;
    robot6axis/arm1RowA/m23 AT 7033 : REAL := 0.0;
    robot6axis/arm1RowA/m24 AT 7034 : REAL := 1.0;
    robot6axis/arm1RowA/m31 AT 7035 : REAL := 0.0;
    robot6axis/arm1RowA/m32 AT 7036 : REAL := 0.0;
    robot6axis/arm1RowA/m33 AT 7037 : REAL := 9.90274;
    robot6axis/arm1RowA/m34 AT 7038 : REAL := -51.6357;
    robot6axis/arm1RowA/m41 AT 7039 : REAL := 0.0;
    robot6axis/arm1RowA/m42 AT 7040 : REAL := 0.0;
    robot6axis/arm1RowA/m43 AT 7041 : REAL := 0.0;
    robot6axis/arm1RowA/m44 AT 7042 : REAL := 1.0;
    robot6axis/arm1RowA/armLengthCalc AT 7043 : REAL := 0.0;
    robot6axis/arm1RowA/functionActiveLocale AT 320 : BOOL := false;
    robot6axis/arm1RowA/product_id AT 676 : DINT := -1;
    robot6axis/arm1RowA/arm_id AT 677 : DINT := -1;
    robot6axis/arm1RowA/timeToGripParam AT 7044 : REAL := 0.15;
    robot6axis/arm1RowA/armLength AT 7045 : REAL := 100.0;
    robot6axis/arm1RowA/armWidth AT 7046 : REAL := 200.0;
    robot6axis/arm1RowA/armHeight AT 7047 : REAL := 5.0;
    robot6axis/arm1RowA/armType AT 678 : INT := 0;
    robot6axis/arm1RowB/armOrigin AT 6597 : ARRAY[1..3] OF REAL := [3(0.0)];
    robot6axis/arm1RowB/overallArmQuatInput AT 6602 : ARRAY[1..4] OF REAL := [4(0.0)];
    robot6axis/arm1RowB/structRotVector AT 98 : ARRAY[1..3] OF REAL := [0.0, 1.0, 0.0];
    robot6axis/arm1RowB/structRotDeg AT 97 : REAL := 90.0;
    robot6axis/arm1RowB/driveRotVector AT 6397 : ARRAY[1..3] OF REAL := [2(0.0), 1.0];
    robot6axis/arm1RowB/driveRotDeg AT 6396 : REAL := 0.0;
    robot6axis/arm1RowB/ownRotDeg AT 6395 : REAL := 0.0;
    robot6axis/arm1RowB/driveResizeLength AT 6394 : REAL := 0.0;
    robot6axis/arm1RowB/functionActive AT 13 : BOOL := false;
    robot6axis/arm1RowB/armExtrem AT 6389 : ARRAY[1..3] OF REAL := [3(0.0)];
    robot6axis/arm1RowB/overallArmRotOutput AT 6383 : ARRAY[1..4] OF REAL := [4(0.0)];
    robot6axis/arm1RowB/productId AT 612 : DINT := -1;
    robot6axis/arm1RowB/status_act_prod AT 679 : DINT := 0;
    robot6axis/arm1RowB/m11 AT 7048 : REAL := 50.0;
    robot6axis/arm1RowB/m12 AT 7049 : REAL := -3.71633e-005;
    robot6axis/arm1RowB/m13 AT 7050 : REAL := 0.000872664;
    robot6axis/arm1RowB/m14 AT 7051 : REAL := 900.92;
    robot6axis/arm1RowB/m21 AT 7052 : REAL := 0.0;
    robot6axis/arm1RowB/m22 AT 7053 : REAL := -200.0;
    robot6axis/arm1RowB/m23 AT 7054 : REAL := -0.00532325;
    robot6axis/arm1RowB/m24 AT 7055 : REAL := 815.446;
    robot6axis/arm1RowB/m31 AT 7056 : REAL := 0.00872665;
    robot6axis/arm1RowB/m32 AT 7057 : REAL := 0.21293;
    robot6axis/arm1RowB/m33 AT 7058 : REAL := -5.0;
    robot6axis/arm1RowB/m34 AT 7059 : REAL := 451.412;
    robot6axis/arm1RowB/m41 AT 7060 : REAL := 0.0;
    robot6axis/arm1RowB/m42 AT 7061 : REAL := 0.0;
    robot6axis/arm1RowB/m43 AT 7062 : REAL := 0.0;
    robot6axis/arm1RowB/m44 AT 7063 : REAL := 1.0;
    robot6axis/arm1RowB/armLengthCalc AT 7064 : REAL := 0.0;
    robot6axis/arm1RowB/functionActiveLocale AT 321 : BOOL := false;
    robot6axis/arm1RowB/product_id AT 680 : DINT := -1;
    robot6axis/arm1RowB/arm_id AT 681 : DINT := -1;
    robot6axis/arm1RowB/timeToGripParam AT 7065 : REAL := 0.15;
    robot6axis/arm1RowB/armLength AT 7066 : REAL := 50.0;
    robot6axis/arm1RowB/armWidth AT 7067 : REAL := 200.0;
    robot6axis/arm1RowB/armHeight AT 7068 : REAL := 5.0;
    robot6axis/arm1RowB/armType AT 682 : INT := 0;
  END_VAR
END_CONFIGURATION
